TYPE DUT_RecipeCommand :
STRUCT
	SkillID: INT;
	SkillName: STRING(80);
	Quantity: LREAL;
END_STRUCT
END_TYPE

(* stored: Version 1.1.0.1, ProductVersion 3.1.0.25
   DUT DUT_RecipeCommand: Id {ae159bd1-87fc-4171-a193-4aa72e80905c} *)
